// TIA Portal V20 export
// export: Created 2026-04-11T06:02:30.3743372Z, ExportSetting WithDefaults, DisplayName Totally Integrated Automation Portal, DisplayVersion V20, DisplayName TIA Portal Openness, DisplayVersion V20, DisplayName TIA Portal Version Control Interface, DisplayVersion V20, DisplayName STEP 7 Professional, DisplayVersion V20, DisplayName STEP 7 Safety, DisplayVersion V20, DisplayName WinCC Basic/Comfort/Advanced, DisplayVersion V20, DisplayName WinCC Unified, DisplayVersion V20
TYPE "udtHMI_3RW44Control"
// stored: IsFailsafeCompliant false
   STRUCT
      iMode : Int;   // Current mode
      iErrorCode { ExternalWritable := 'False'} : Int;   // Error code
      iStatus { ExternalWritable := 'False'} : Int;   // Status for HMI display
      iParameterSet : Int := 1;   // Parameter Set (Configured on 3RW44: 1, 2 or 3, default 1)
      bPB_ResetError : Bool;   // PB Reset block errors
      bPB_CW : Bool;   // PB Move CW in manual mode
      bPB_CCW : Bool;   // PB Move CCW in manual mode
      bPB_Stop : Bool;   // PB Stop in manual mode
      bPB_EmergencyStart : Bool;   // PB Emergency Start
      bPBEN_ResetError { ExternalWritable := 'False'} : Bool;   // PB Reset error enabled
      bPBEN_CW { ExternalWritable := 'False'} : Bool;   // PB CW enabled
      bPBEN_CCW { ExternalWritable := 'False'} : Bool;   // PB CCW enabled
      bPBEN_Stop { ExternalWritable := 'False'} : Bool;   // PB Stop enabled
      bPBEN_EmergencyStart { ExternalWritable := 'False'} : Bool;   // PB Emergency Start Enabled
      bSlowSpeedOn : Bool;   // Slow Speed Enabled
      bQuickStopDisabled : Bool;   // Quick Stop Function Disabled
      bEmergencyStartActive { ExternalWritable := 'False'} : Bool;   // Emergency Start Active
      bCWOn { ExternalWritable := 'False'} : Bool;   // Moving CW
      bCCWOn { ExternalWritable := 'False'} : Bool;   // Moving CCW
      bRampOperation { ExternalWritable := 'False'} : Bool;   // True when ramping up/down (inverse of signal bypass on 3RW30/40)
      bSignalRun { ExternalWritable := 'False'} : Bool;   // Run signal
      bError { ExternalWritable := 'False'} : Bool;   // Overall error
      bInterlock { ExternalWritable := 'False'} : Bool;   // Motor interlocked
      rActualCurrent { ExternalWritable := 'False'} : Real;   // Current Output from 3RW44
      bShowOptions : Bool;   // Needed for WinCC Pro Popup to show/hide options
   END_STRUCT;
END_TYPE
